(*Take Individual time elements of a TIMESTRUCT and create a TOD type return
	author: Brent Lekx-Toniolo Of Sodecia GTAC
	date: May 2016
	version 1.0
		- initial concept


	Last Edit: 27-May-2016, blt
*)

FUNCTION FUN_GTAC_TIMESTRUCTtoTOD : TOD
VAR_INPUT
	TIMESTRUCT: TIMESTRUCT;

END_VAR
VAR
	Hours_as_MS: UDINT;
	Minutes_as_MS: UDINT;
	Seconds_as_MS: UDINT;
	Milliseconds_as_MS: UDINT;
END_VAR

(*Calculate Millsecond Value of each OTSTRUCT Element*)

	Hours_as_MS:= TIMESTRUCT.wHour * 3600000;
	Minutes_as_MS:= TIMESTRUCT.wMinute * 60000;
	Seconds_as_MS:= TIMESTRUCT.wSecond * 1000;
	Milliseconds_as_MS:= TIMESTRUCT.wMilliseconds;

(*Return Total Value in Milliseconds, this is TOD*)

	FUN_GTAC_TIMESTRUCTtoTOD:= UDINT_TO_TOD(Hours_As_MS + Minutes_As_MS + Seconds_As_MS + Milliseconds_As_MS);

END_FUNCTION

(* stored: Version 1.1.0.1, ProductVersion 3.1.4024.5
   POU FUN_GTAC_TIMESTRUCTtoTOD: Id {7a96b2b7-6a4a-436e-b540-2706fc9d8fad}, SpecialFunc None *)
